FUNCTION_BLOCK X20DO4623 (* Service Interface Function Block Type *)
  (* Standard: 61499-2; Description: Copyright (c) 2011 AIT This program and the accompanying materials are made available under the terms of the Eclipse Public License 2.0 which is available at https://www.eclipse.org/legal/epl-2.0/ SPDX-License-Identifier: EPL-2.0 *)
  (* Version 3.0, 2025-04-14, Patrick Aigner, changed package *)
  (* Version 1.0, 2011-05-31, Filip Andren, Thomas Strasser, AIT *)
  (* Version 0.0, 2011-05-31, Filip Andren, AIT *)
  PACKAGE powerlink;
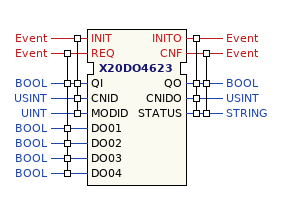
  EVENT_INPUT
    INIT WITH QI, CNID, MODID; (* Service Initialization *)
    REQ WITH DO01, DO02, DO03, DO04, QI; (* Service Request *)
  END_EVENT
  EVENT_OUTPUT
    INITO WITH QO, STATUS, CNIDO; (* Initialization Confirm *)
    CNF WITH STATUS, QO; (* Confirmation of Requested Service *)
  END_EVENT
  VAR_INPUT
    QI : BOOL; (* Event Input Qualifier *)
    CNID : USINT; (* Client Node ID *)
    MODID : UINT; (* Station Number *)
    DO01 : BOOL; (* Digital Output 01 *)
    DO02 : BOOL; (* Digital Output 02 *)
    DO03 : BOOL; (* Digital Output 03 *)
    DO04 : BOOL; (* Digital Output 04 *)
  END_VAR
  VAR_OUTPUT
    QO : BOOL; (* Event Output Qualifier *)
    CNIDO : USINT; (* Client Node ID Output *)
    STATUS : STRING; (* Service Status *)
  END_VAR
  SERVICE APPLICATION/RESOURCE
    SEQUENCE normal_establishment
      APPLICATION.INIT+(PARAMS) -> APPLICATION.INITO+(PARAMS);
    END_SEQUENCE
    SEQUENCE unsuccessful_establishment
      APPLICATION.INIT+(PARAMS) -> APPLICATION.INITO-(STATUS);
    END_SEQUENCE
    SEQUENCE request_confirm
      APPLICATION.REQ+(SD) -> APPLICATION.CNF+(RD);
    END_SEQUENCE
    SEQUENCE request_inhibited
      APPLICATION.REQ-(SD) -> APPLICATION.CNF-(STATUS);
    END_SEQUENCE
    SEQUENCE request_error
      APPLICATION.REQ+(SD) -> APPLICATION.CNF-(STATUS);
    END_SEQUENCE
    SEQUENCE indication_response
      RESOURCE.indicate(RD) -> APPLICATION.IND+(RD);
      APPLICATION.RSP(QI,SD) -> RESOURCE.response(QI,SD);
    END_SEQUENCE
    SEQUENCE indication_inhibited
      RESOURCE.indicate(RD,QI=FALSE) -> RESOURCE.inhibited();
    END_SEQUENCE
    SEQUENCE error_indication
      RESOURCE.error(STATUS) -> APPLICATION.IND-(STATUS);
    END_SEQUENCE
    SEQUENCE application_initiated_termination
      APPLICATION.INIT-() -> APPLICATION.INITO-(STATUS);
    END_SEQUENCE
    SEQUENCE resource_initiated_termination
      -> APPLICATION.INITO-(STATUS);
    END_SEQUENCE
  END_SERVICE
END_FUNCTION_BLOCK
